(* CODESYS project e!C_SmartCoupler_Test_1.ecp

Project tree, tasks and I/O mapping:
  Generic_MODBUS_Master : ThirdParty Modbus Master, WAGO, order no. GenericModbusMaster, version 1.0.0.1
  PFCx00_SmartCoupler : 750-8202 PFC200 2ETH RS, WAGO, order no. 0750-8202, version 5.13.2.22
    application PFCx00_SmartCoupler
      libraries: ; VisuDialogs, * (System); WagoTypesCommon, 1.5.3.0 (WAGO); WagoAppHART, 1.7.1.0 (WAGO); WagoAppSolenoid, 1.7.1.0 (WAGO); WagoAppPowerMeasurement, 1.7.1.0 (WAGO); WagoTypesCom, 1.6.1.0 (WAGO); WagoAppDALI, 1.3.0.0 (WAGO); WagoSysKbusModule, 1.8.2.0 (WAGO); AnyViz Cloud Adapter, 1.4.0.0 (Mirasoft GmbH & Co. KG); WagoSysKbusServices, 1.8.7.0 (WAGO); WagoAppPlcModbus, 1.1.2.0 (WAGO); WagoTypesAsync_Internal_Template, 1.0.0.1 (WAGO); WagoSysModule_75x_632, 1.8.1.0 (WAGO); WagoSysModule_75x_48x, 1.5.1.0 (WAGO); WagoVisuIcons, 1.0.1.0 (WAGO); WagoSysModule_75x_49x, 1.7.1.0 (WAGO); WagoSysModule_753_647, 1.1.1.0 (WAGO); WagoAppKNX, 1.0.4.0 (WAGO)
      task Cloud_Task (freewheeling, priority 15) calls Cloud
      task PLC_Task (cyclic, interval t#10ms, priority 12) calls PLC_PRG
      task VISU_TASK (cyclic, interval 100 ms, priority 14) calls VisuElems.Visu_Prg
      program PLC_PRG [ST]
      GlobalData/
        global variables GCL_SmartCoupler
        global variables GVL_SmartCoupler
      Symbols
      visualisation Visualization
      program Cloud [ST]
    Kbus : Kbus, WAGO, version 1.4.0.2
        unmapped channels: K-BUS diagnostics
    MODBUS
      MODBUS : MODBUS, WAGO, order no. n/a, version 1.1.1.15
        LocalDeviceModbus : MODBUS Slave, WAGO, order no. n/a, version 1.1.1.15
          TcpSettings : Modbus TCP Slave, WAGO, order no. n/a, version 1.1.1.15
              settings: TCP Port = 503; TCP connection watchdog = 200 10ms
          UdpSettings : Modbus UDP Slave, WAGO, order no. n/a, version 1.1.1.15
              settings: UDP Port = 503
    Serial
      COM1 : COM1, WAGO, version 0.0.0.19
  libraries: WagoAppPlcModbus, * (WAGO); WagoAppHART, * (WAGO); WagoAppSolenoid, * (WAGO); WagoAppPowerMeasurement, * (WAGO); WagoTypesCom, * (WAGO); WagoTypesCommon, * (WAGO); WagoAppDALI, * (WAGO); VisuSymbols, 3.5.10.0 (System); WagoSysKbusModule, * (WAGO); WagoAppKNX, 1.0.4.0 (WAGO); WagoSysKbusServices, 1.8.7.0 (WAGO); WagoTypesAsync_Internal_Template, 1.0.0.1 (WAGO); WagoSysModule_75x_632, 1.8.1.0 (WAGO); WagoSysModule_75x_48x, 1.5.1.0 (WAGO); WagoVisuIcons, 1.0.1.0 (WAGO); WagoSysModule_75x_49x, 1.7.1.0 (WAGO); WagoSysModule_753_647, 1.1.1.0 (WAGO)
  GlobalStruct/
    data type DUT_WordAndBytes
    data type DUT_ModuleDataAccess
    data type DUT_RealAndBytes
    data type DUT_ModuleFunctionAccess
    data type DUT_ModuleDescriptor
    data type DUT_ModuleInterface
  GlobalProgram/
    program SmartCoupler [ST]: DrivePMeasurementModuleAccess, DriveSimpleDIOModuleAccess, DriveSolenoidModuleAccess, DriveHartModuleAccess, InitModuleDescriptor, DriveDaliModuleAccess, DriveSimpleAIOModuleAccess, DriveKnxModuleAccess
    program ModbusSlave [ST]: MapModbusData
  text list GlobalTextList
*)

// GlobalStruct/DUT_WordAndBytes
TYPE DUT_WordAndBytes :
UNION
	wValue: WORD;
	abValue: ARRAY[0..1] OF BYTE;	
END_UNION
END_TYPE

// GlobalStruct/DUT_ModuleDataAccess
TYPE DUT_ModuleDataAccess :
STRUCT
	sModuleList: STRING;
	udiModuleID: UDINT;
	auiOrderNumber: ARRAY[0..3] OF UINT;
	uiModuleChannels: UINT;
	uiModuleType: UINT;
	uiModulePiSize: UINT;
	uiModulePiInputSize: UINT;
	uiModulePiOutputSize: UINT;
	wModuleOutput_Data_1: WORD;
	wModuleOutput_Data_2: WORD;
	wModuleOutput_Data_3: WORD;
	wModuleOutput_Data_4: WORD;
	wModuleOutput_Data_5: WORD;
	wModuleOutput_Data_6: WORD;
	wModuleOutput_Data_7: WORD;
	wModuleOutput_Data_8: WORD;
	wModuleOutput_Data_9: WORD;
	wModuleOutput_Data_10: WORD;
	wModuleOutput_Data_11: WORD;
	wModuleOutput_Data_12: WORD;
	wModuleOutput_Data_13: WORD;
	wModuleOutput_Data_14: WORD;
	wModuleOutput_Data_15: WORD;
	wModuleOutput_Data_16: WORD;
	wModuleInput_Data_1: WORD;
	wModuleInput_Data_2: WORD;
	wModuleInput_Data_3: WORD;
	wModuleInput_Data_4: WORD;
	wModuleInput_Data_5: WORD;
	wModuleInput_Data_6: WORD;
	wModuleInput_Data_7: WORD;
	wModuleInput_Data_8: WORD;
	wModuleInput_Data_9: WORD;
	wModuleInput_Data_10: WORD;
	wModuleInput_Data_11: WORD;
	wModuleInput_Data_12: WORD;
	wModuleInput_Data_13: WORD;
	wModuleInput_Data_14: WORD;
	wModuleInput_Data_15: WORD;
	wModuleInput_Data_16: WORD;
	pawModuleOutput: POINTER TO ARRAY[1..GCL_SmartCoupler.LIM_OF_IO_FRAME] OF WORD;
	pawModuleInput: POINTER TO ARRAY[1..GCL_SmartCoupler.LIM_OF_IO_FRAME] OF WORD;
END_STRUCT
END_TYPE

// GlobalStruct/DUT_RealAndBytes
TYPE DUT_RealAndBytes :
UNION
	rValue: REAL;
	dwValue: DWORD;
	awValue: ARRAY[0..1] OF WORD;
	abValue: ARRAY[0..3] OF BYTE;
END_UNION
END_TYPE

// GlobalStruct/DUT_ModuleFunctionAccess
TYPE DUT_ModuleFunctionAccess :
STRUCT
	FbAC_Compact_494: WagoAppPowerMeasurement.FbAC_Compact_494;
	FbAC_Compact_495: WagoAppPowerMeasurement.FbAC_Compact_495;
	FbSolenoidBasicControl: WagoAppSolenoid.FbBasicControl;
	FbKnxMaster_TM: WagoAppKnx.FbKNX_Master_TM;
	FbDaliMaster: WagoAppDali.FbDaliMaster;
	FbDaliSendDimValue: WagoAppDali.FbDaliSendDimValue;
	FbHART_Current: WagoAppHart.FbHART_Current := (xEnable := TRUE);
	FbHART_CMD3_1: WagoAppHart.FbHART_CMD3;
	FbHART_CMD3_2: WagoAppHart.FbHART_CMD3;
	xHartReadTrigger_1: BOOL;
	xHartReadTrigger_2: BOOL;
	wHartChannelSchedule: WORD;
	TON_HartScheduleDelay: TON;
	TOF_HartCmdMonitor_1: TOF;
	TOF_HartCmdMonitor_2: TOF;
	tHartScheduleDelay: TIME := T#2S;
	tHartCmdMonitorTimeout: TIME := T#5S;
	iHartGenericErrorCnt: INT;
	iHartCmdErrorCnt_1: INT;
	iHartCmdErrorCnt_2: INT;
END_STRUCT
END_TYPE

// GlobalStruct/DUT_ModuleDescriptor
TYPE DUT_ModuleDescriptor :
STRUCT
	pDUT_ModuleInterface: POINTER TO DUT_ModuleInterface;
	pDUT_ModuleAccess: POINTER TO DUT_ModuleDataAccess;	
	pDUT_FunctionAccess: POINTER TO DUT_ModuleFunctionAccess;
END_STRUCT
END_TYPE

// GlobalStruct/DUT_ModuleInterface
TYPE DUT_ModuleInterface :
STRUCT
	FbModuleProcessInputsOutputs: WagoSysKbusModule.FbModuleProcessInputsOutputs;
	FbModule_75x_632: WagoSysKbusModule.FbModule_75x_632;
	FbModule_753_646: WagoSysKbusModule.FbModule_753_646;
	FbModule_753_647: WagoSysKbusModule.FbModule_753_647;
	FbModule_75x_48x: WagoSysKbusModule.FbModule_75x_48x;
	FbModule_75x_494: WagoSysKbusModule.FbModule_75x_494;
	FbModule_75x_495: WagoSysKbusModule.FbModule_75x_495;
(*
	FbModule_75x_632: WagoSysKbusModule.WagoSysModule_75x_632.FbModule_75x_632;
	FbModule_753_646: WagoSysKbusModule.WagoSysModule_753_646.FbModule_753_646;
	FbModule_753_647: WagoSysKbusModule.WagoSysModule_753_647.FbModule_753_647;
	FbModule_75x_48x: WagoSysKbusModule.WagoSysModule_75x_48x.FbModule_75x_48x;
	FbModule_75x_494: WagoSysKbusModule.WagoSysModule_75x_49x.FbModule_75x_494;
	FbModule_75x_495: WagoSysKbusModule.WagoSysModule_75x_49x.FbModule_75x_495;
*)
END_STRUCT
END_TYPE

// PFCx00_SmartCoupler/PFCx00_SmartCoupler/GlobalData/GCL_SmartCoupler
{attribute 'qualified_only'}
VAR_GLOBAL CONSTANT
	LIM_OF_IO_MODULES: INT := 64;
	LIM_OF_IO_SEGMENT: INT := 4096;
	LIM_OF_IO_FRAME: USINT := 16; (* Number of WORD per module *)
END_VAR

// PFCx00_SmartCoupler/PFCx00_SmartCoupler/GlobalData/GVL_SmartCoupler
{attribute 'qualified_only'}
VAR_GLOBAL
	aDUT_ModuleDescriptor: ARRAY[1..GCL_SmartCoupler.LIM_OF_IO_MODULES] OF DUT_ModuleDescriptor;
	aDUT_ModuleInterface: ARRAY[1..GCL_SmartCoupler.LIM_OF_IO_MODULES] OF DUT_ModuleInterface;
	aDUT_ModuleDataAccess: ARRAY[1..GCL_SmartCoupler.LIM_OF_IO_MODULES] OF DUT_ModuleDataAccess;
	aDUT_ModuleFunctionAccess: ARRAY[1..GCL_SmartCoupler.LIM_OF_IO_MODULES] OF DUT_ModuleFunctionAccess;	
	awModuleInputData: ARRAY[1..GCL_SmartCoupler.LIM_OF_IO_SEGMENT] OF WORD;
	awModuleOutputData: ARRAY[1..GCL_SmartCoupler.LIM_OF_IO_SEGMENT] OF WORD;
	DUT_ModuleData: DUT_RealAndBytes;
	bModule646Index: BYTE;
	bModule647Index: BYTE;
END_VAR

// PFCx00_SmartCoupler/PFCx00_SmartCoupler/Cloud
PROGRAM Cloud
VAR
	AnyVizClient: AnyVizClient := (ProjectID := 324, Password := 'wago1234');
	Status: STRING(255);
	Error: BOOL;
	Connected: BOOL;
END_VAR


(*
AnyVizClient(
	Status				=> Status, 
	Error				=> Error, 
	Connected			=> Connected);
*)

END_PROGRAM

// PFCx00_SmartCoupler/PFCx00_SmartCoupler/PLC_PRG
PROGRAM PLC_PRG
VAR

END_VAR



ModbusSlave();
SmartCoupler();

END_PROGRAM

// GlobalProgram/ModbusSlave
PROGRAM ModbusSlave
VAR
	FbMbSimpleServerUdp: FbMbSimpleServerUdp;
	FbMbSimpleServerTcp: FbMbSimpleServerTcp;
	xMbTcpOpen: BOOL := TRUE;
	wMbTcpPort: WORD := 502;
	utMbTcpKeepAlive: typKeepAlive;
	xMbTcpIsOpen: BOOL;
	xMbTcpError: BOOL;
	oMbTcpStatus: WagoSysErrorBase.FbResult;
	udiMbTcpConnectedClients: UDINT;
	bMbTcpUnitId: BYTE := 1;
	axMbDiscreteInputs: ARRAY[0..0] OF BOOL;
	axMbCoils: ARRAY[0..0] OF BOOL;
	oMbTcpAccessInfo: FbMbAccessInfo;
	xMbUdpOpen: BOOL := TRUE;
	wMbUdpPort: WORD := 502;
	xMbUdpIsOpen: BOOL;
	xMbUdpError: BOOL;
	oMbUdpStatus: WagoSysErrorBase.FbResult;
	bMbUdpUnitId: BYTE := 1;
	oMbUdpAccessInfo: FbMbAccessInfo;
	FbMbSimpleServerSerial: FbMbSimpleServerSerial;
	xMbRtuConnect: BOOL := TRUE;
	udiMbRtuBaudrate: UDINT := 19200;
	usiMbRtuDataBits: USINT := 8;
	eMbRtuParity: WagoTypesCom.eTTYParity := ETTYPARITY.None;
	eMbRtuStopBits: WagoTypesCom.eTTYStopBits := ETTYSTOPBITS.one;
	eMbRtuHandshake: WagoTypesCom.eTTYHandshake := ETTYHANDSHAKE.None;
	eMbRtuPhysical: WagoTypesCom.eTTYPhysicalLayer := ETTYPHYSICALLAYER.RS485_HalfDuplex;
	eMbRtuFrameType: eMbFrameType := EMBFRAMETYPE.RTU;
	xMbRtuIsConnected: BOOL;
	xMbRtuError: BOOL;
	oMbRtuStatus: WagoSysErrorBase.FbResult;
	bMbRtuUnitId: BYTE := 1;
	oMbRtuAccessInfo: FbMbAccessInfo;
END_VAR


FbMbSimpleServerTcp(
	xOpen				:= xMbTcpOpen, 
	wPort				:= wMbTcpPort, 
	utKeepAlive			:= utMbTcpKeepAlive, 
	xIsOpen				=> xMbTcpIsOpen, 
	xError				=> xMbTcpError, 
	oStatus				=> oMbTcpStatus, 
	udiConnectedClients	=> udiMbTcpConnectedClients, 
	bUnitId				:= bMbTcpUnitId, 
	axDiscreteInputs	:= axMbDiscreteInputs, 
	axCoils				:= axMbCoils, 
	awInputRegisters	:= GVL_SmartCoupler.awModuleInputData, 
	awHoldingRegisters	:= GVL_SmartCoupler.awModuleOutputData, 
	oMbAccessInfo		=> oMbTcpAccessInfo);

FbMbSimpleServerUdp(
	xOpen				:= xMbUdpOpen, 
	wPort				:= wMbUdpPort, 
	xIsOpen				=> xMbUdpIsOpen, 
	xError				=> xMbUdpError, 
	oStatus				=> oMbUdpStatus, 
	bUnitId				:= bMbUdpUnitId, 
	axDiscreteInputs	:= axMbDiscreteInputs, 
	axCoils				:= axMbCoils, 
	awInputRegisters	:= GVL_SmartCoupler.awModuleInputData, 
	awHoldingRegisters	:= GVL_SmartCoupler.awModuleOutputData, 
	oMbAccessInfo		=> oMbUdpAccessInfo);

FbMbSimpleServerSerial(
	xConnect			:= xMbRtuConnect, 
	I_Port				:= COM1, 
	udiBaudrate			:= udiMbRtuBaudrate, 
	usiDataBits			:= usiMbRtuDataBits, 
	eParity				:= eMbRtuParity, 
	eStopBits			:= eMbRtuStopBits, 
	eHandshake			:= eMbRtuHandshake, 
	ePhysical			:= eMbRtuPhysical, 
	eFrameType			:= eMbRtuFrameType, 
	xIsConnected		=> xMbRtuIsConnected, 
	xError				=> xMbRtuError, 
	oStatus				=> oMbRtuStatus, 
	bUnitId				:= bMbRtuUnitId, 
	axDiscreteInputs	:= axMbDiscreteInputs, 
	axCoils				:= axMbCoils, 
	awInputRegisters	:= GVL_SmartCoupler.awModuleInputData, 
	awHoldingRegisters	:= GVL_SmartCoupler.awModuleOutputData, 
	oMbAccessInfo		=> oMbRtuAccessInfo);

ACTION MapModbusData:

;
END_ACTION

END_PROGRAM

// GlobalProgram/SmartCoupler
PROGRAM SmartCoupler
VAR
	I_Terminal: WagoSysModuleBase.WagoTypesModuleBase.I_TerminalBase;
	FBTerminalManagerResult: FBResult;
	xTerminalInit: BOOL;
	usiModuleIndex: USINT;
	uiModuleMapIndex: UINT;
	usiModuleIndexLimit: USINT;
	uiChannelIndex: UINT;
END_VAR


IF  (TerminalManager.isBusInit(WagoTypesBusServices.eBusType.KBUS) = TRUE) THEN
	IF (xTerminalInit = FALSE) THEN
		usiModuleIndexLimit := TerminalManager.getTerminalQuantity(WagoSysKbusModule.KBUS);
	END_IF
	uiModuleMapIndex := 1;
	GVL_SmartCoupler.bModule646Index := 1;
	GVL_SmartCoupler.bModule647Index := 1;
	FOR usiModuleIndex := 1 TO usiModuleIndexLimit DO
		GVL_SmartCoupler.aDUT_ModuleDescriptor[usiModuleIndex].pDUT_ModuleInterface := ADR(GVL_SmartCoupler.aDUT_ModuleInterface[usiModuleIndex]);
		GVL_SmartCoupler.aDUT_ModuleDescriptor[usiModuleIndex].pDUT_ModuleAccess := ADR(GVL_SmartCoupler.aDUT_ModuleDataAccess[usiModuleIndex]);
		GVL_SmartCoupler.aDUT_ModuleDescriptor[usiModuleIndex].pDUT_FunctionAccess := ADR(GVL_SmartCoupler.aDUT_ModuleFunctionAccess[usiModuleIndex]);
		IF (xTerminalInit = FALSE) THEN
			InitModuleDescriptor();
		ELSE
	
			(* Data exchange for Address-based fieldbus interface/gateway, e.g. Modbus *)
			GVL_SmartCoupler.aDUT_ModuleDataAccess[usiModuleIndex].pawModuleInput := ADR(GVL_SmartCoupler.awModuleInputData[uiModuleMapIndex]);
			GVL_SmartCoupler.aDUT_ModuleDataAccess[usiModuleIndex].pawModuleOutput := ADR(GVL_SmartCoupler.awModuleOutputData[uiModuleMapIndex]);

			(* Data exchange for Symbol-based fieldbus interface/gateway, e.g. OPCUA *)
			(*
			GVL_SmartCoupler.aDUT_ModuleDataAccess[usiModuleIndex].pawModuleInput := ADR(GVL_SmartCoupler.aDUT_ModuleDataAccess[usiModuleIndex].wModuleInput_Data_1);
			GVL_SmartCoupler.aDUT_ModuleDataAccess[usiModuleIndex].pawModuleOutput := ADR(GVL_SmartCoupler.aDUT_ModuleDataAccess[usiModuleIndex].wModuleOutput_Data_1);
			*)
			CASE GVL_SmartCoupler.aDUT_ModuleDataAccess[usiModuleIndex].uiModuleType OF
	
				COMPLEX_INPUT, COMPLEX_OUTPUT:
					DriveSimpleAIOModuleAccess();
				COMPLEX_INOUT:
					CASE GVL_SmartCoupler.aDUT_ModuleDataAccess[usiModuleIndex].auiOrderNumber[1] OF
						482, 484:
							DriveHartModuleAccess();
						494, 495:
							DrivePMeasurementModuleAccess();
						632:
							DriveSolenoidModuleAccess();
						646:
							DriveKnxModuleAccess();
							GVL_SmartCoupler.bModule646Index := GVL_SmartCoupler.bModule646Index + 1;
						647:
							DriveDaliModuleAccess();
							GVL_SmartCoupler.bModule647Index := GVL_SmartCoupler.bModule647Index + 1;
					END_CASE
				DIGITAL_INPUT, DIGITAL_INPUT_DIAG, DIGITAL_OUTPUT, DIGITAL_OUTPUT_DIAG, DIGITAL_INOUT, DIGITAL_INOUT_DIAG, DIGITAL_DIAG:
					DriveSimpleDIOModuleAccess();
	
			END_CASE
			uiModuleMapIndex := uiModuleMapIndex + GCL_SmartCoupler.LIM_OF_IO_FRAME;
		END_IF
	END_FOR
	xTerminalInit := TRUE;
END_IF

ACTION DrivePMeasurementModuleAccess:

IF (GVL_SmartCoupler.aDUT_ModuleDataAccess[usiModuleIndex].uiModuleType = 494) THEN
	GVL_SmartCoupler.aDUT_ModuleFunctionAccess[usiModuleIndex].FbAC_Compact_494.xEnable (*:= WORD_TO_BOOL(GVL_SmartCoupler.aDUT_ModuleDataAccess[usiModuleIndex].pawModuleOutput^[1])*);
	GVL_SmartCoupler.aDUT_ModuleFunctionAccess[usiModuleIndex].FbAC_Compact_494.tCycleTime (*:= WORD_TO_TIME(GVL_SmartCoupler.aDUT_ModuleDataAccess[usiModuleIndex].pawModuleOutput^[2])*);
	GVL_SmartCoupler.aDUT_ModuleFunctionAccess[usiModuleIndex].FbAC_Compact_494.rSelectedScalingFactor (*:= WORD_TO_REAL(GVL_SmartCoupler.aDUT_ModuleDataAccess[usiModuleIndex].pawModuleOutput^[3])*);	
	GVL_SmartCoupler.aDUT_ModuleFunctionAccess[usiModuleIndex].FbAC_Compact_494(I_Port := GVL_SmartCoupler.aDUT_ModuleInterface[usiModuleIndex].FbModule_75x_494);
	GVL_SmartCoupler.DUT_ModuleData.rValue := GVL_SmartCoupler.aDUT_ModuleFunctionAccess[usiModuleIndex].FbAC_Compact_494.aVoltage_L_N[1];
	GVL_SmartCoupler.aDUT_ModuleDataAccess[usiModuleIndex].pawModuleInput^[1] := GVL_SmartCoupler.DUT_ModuleData.awValue[0];
	GVL_SmartCoupler.aDUT_ModuleDataAccess[usiModuleIndex].pawModuleInput^[2] := GVL_SmartCoupler.DUT_ModuleData.awValue[1];
	GVL_SmartCoupler.DUT_ModuleData.rValue := GVL_SmartCoupler.aDUT_ModuleFunctionAccess[usiModuleIndex].FbAC_Compact_494.aVoltage_L_N[2];
	GVL_SmartCoupler.aDUT_ModuleDataAccess[usiModuleIndex].pawModuleInput^[3] := GVL_SmartCoupler.DUT_ModuleData.awValue[0];
	GVL_SmartCoupler.aDUT_ModuleDataAccess[usiModuleIndex].pawModuleInput^[4] := GVL_SmartCoupler.DUT_ModuleData.awValue[1];
	GVL_SmartCoupler.DUT_ModuleData.rValue := GVL_SmartCoupler.aDUT_ModuleFunctionAccess[usiModuleIndex].FbAC_Compact_494.aVoltage_L_N[3];
	GVL_SmartCoupler.aDUT_ModuleDataAccess[usiModuleIndex].pawModuleInput^[5] := GVL_SmartCoupler.DUT_ModuleData.awValue[0];
	GVL_SmartCoupler.aDUT_ModuleDataAccess[usiModuleIndex].pawModuleInput^[6] := GVL_SmartCoupler.DUT_ModuleData.awValue[1];
ELSIF (GVL_SmartCoupler.aDUT_ModuleDataAccess[usiModuleIndex].uiModuleType = 495) THEN
	GVL_SmartCoupler.aDUT_ModuleFunctionAccess[usiModuleIndex].FbAC_Compact_495.xEnable (*:= WORD_TO_BOOL(GVL_SmartCoupler.aDUT_ModuleDataAccess[usiModuleIndex].pawModuleOutput^[1])*);
	GVL_SmartCoupler.aDUT_ModuleFunctionAccess[usiModuleIndex].FbAC_Compact_495.tCycleTime (*:= WORD_TO_TIME(GVL_SmartCoupler.aDUT_ModuleDataAccess[usiModuleIndex].pawModuleOutput^[2])*);
	GVL_SmartCoupler.aDUT_ModuleFunctionAccess[usiModuleIndex].FbAC_Compact_495.rSelectedScalingFactor (*:= WORD_TO_REAL(GVL_SmartCoupler.aDUT_ModuleDataAccess[usiModuleIndex].pawModuleOutput^[3])*);
	GVL_SmartCoupler.aDUT_ModuleFunctionAccess[usiModuleIndex].FbAC_Compact_495(I_Port := GVL_SmartCoupler.aDUT_ModuleInterface[usiModuleIndex].FbModule_75x_495);
	GVL_SmartCoupler.DUT_ModuleData.rValue := GVL_SmartCoupler.aDUT_ModuleFunctionAccess[usiModuleIndex].FbAC_Compact_495.aVoltage_L_N[1];
	GVL_SmartCoupler.aDUT_ModuleDataAccess[usiModuleIndex].pawModuleInput^[1] := GVL_SmartCoupler.DUT_ModuleData.awValue[0];
	GVL_SmartCoupler.aDUT_ModuleDataAccess[usiModuleIndex].pawModuleInput^[2] := GVL_SmartCoupler.DUT_ModuleData.awValue[1];
	GVL_SmartCoupler.DUT_ModuleData.rValue := GVL_SmartCoupler.aDUT_ModuleFunctionAccess[usiModuleIndex].FbAC_Compact_495.aVoltage_L_N[2];
	GVL_SmartCoupler.aDUT_ModuleDataAccess[usiModuleIndex].pawModuleInput^[3] := GVL_SmartCoupler.DUT_ModuleData.awValue[0];
	GVL_SmartCoupler.aDUT_ModuleDataAccess[usiModuleIndex].pawModuleInput^[4] := GVL_SmartCoupler.DUT_ModuleData.awValue[1];
	GVL_SmartCoupler.DUT_ModuleData.rValue := GVL_SmartCoupler.aDUT_ModuleFunctionAccess[usiModuleIndex].FbAC_Compact_495.aVoltage_L_N[3];
	GVL_SmartCoupler.aDUT_ModuleDataAccess[usiModuleIndex].pawModuleInput^[5] := GVL_SmartCoupler.DUT_ModuleData.awValue[0];
	GVL_SmartCoupler.aDUT_ModuleDataAccess[usiModuleIndex].pawModuleInput^[6] := GVL_SmartCoupler.DUT_ModuleData.awValue[1];
END_IF
END_ACTION

ACTION DriveSimpleDIOModuleAccess:

FOR uiChannelIndex := 0 TO GVL_SmartCoupler.aDUT_ModuleDataAccess[usiModuleIndex].uiModuleChannels DO
	IF (GVL_SmartCoupler.aDUT_ModuleDataAccess[usiModuleIndex].uiModulePiInputSize > 0) THEN
		GVL_SmartCoupler.aDUT_ModuleDataAccess[usiModuleIndex].pawModuleInput^[uiChannelIndex+1] :=
			BOOL_TO_WORD(
				GVL_SmartCoupler.aDUT_ModuleInterface[usiModuleIndex].FbModuleProcessInputsOutputs.GetProcessInBit(
							ByteNo	:= 0,
							BitNo	:= UINT_TO_USINT(uiChannelIndex)));
	END_IF
	IF (GVL_SmartCoupler.aDUT_ModuleDataAccess[usiModuleIndex].uiModulePiOutputSize > 0) THEN
		GVL_SmartCoupler.aDUT_ModuleInterface[usiModuleIndex].FbModuleProcessInputsOutputs.SetProcessOutBit(
			ByteNo	:= 0,
			BitNo	:= UINT_TO_USINT(uiChannelIndex),
			OutData	:= WORD_TO_BOOL(GVL_SmartCoupler.aDUT_ModuleDataAccess[usiModuleIndex].pawModuleOutput^[uiChannelIndex+1]));
	END_IF
END_FOR
END_ACTION

ACTION DriveSolenoidModuleAccess:

GVL_SmartCoupler.aDUT_ModuleFunctionAccess[usiModuleIndex].FbSolenoidBasicControl.bSolenoidNo := WORD_TO_BYTE(GVL_SmartCoupler.aDUT_ModuleDataAccess[usiModuleIndex].pawModuleOutput^[1]);
GVL_SmartCoupler.aDUT_ModuleFunctionAccess[usiModuleIndex].FbSolenoidBasicControl.xPowerEnable := WORD_TO_BOOL(GVL_SmartCoupler.aDUT_ModuleDataAccess[usiModuleIndex].pawModuleOutput^[2]);
GVL_SmartCoupler.aDUT_ModuleFunctionAccess[usiModuleIndex].FbSolenoidBasicControl.xCurrentEnable := WORD_TO_BOOL(GVL_SmartCoupler.aDUT_ModuleDataAccess[usiModuleIndex].pawModuleOutput^[3]);
GVL_SmartCoupler.aDUT_ModuleFunctionAccess[usiModuleIndex].FbSolenoidBasicControl.xDitherEnable := WORD_TO_BOOL(GVL_SmartCoupler.aDUT_ModuleDataAccess[usiModuleIndex].pawModuleOutput^[4]);
GVL_SmartCoupler.aDUT_ModuleFunctionAccess[usiModuleIndex].FbSolenoidBasicControl.iCurrent := WORD_TO_INT(GVL_SmartCoupler.aDUT_ModuleDataAccess[usiModuleIndex].pawModuleOutput^[5]);

GVL_SmartCoupler.aDUT_ModuleFunctionAccess[usiModuleIndex].FbSolenoidBasicControl(I_Port := GVL_SmartCoupler.aDUT_ModuleInterface[usiModuleIndex].FbModule_75x_632);

IF (GVL_SmartCoupler.aDUT_ModuleFunctionAccess[usiModuleIndex].FbSolenoidBasicControl.bSolenoidNo = 1) THEN
	GVL_SmartCoupler.aDUT_ModuleDataAccess[usiModuleIndex].pawModuleInput^[1] := INT_TO_WORD(GVL_SmartCoupler.aDUT_ModuleFunctionAccess[usiModuleIndex].FbSolenoidBasicControl.iActualCurrent);
	GVL_SmartCoupler.aDUT_ModuleDataAccess[usiModuleIndex].pawModuleInput^[2] := BOOL_TO_WORD(GVL_SmartCoupler.aDUT_ModuleFunctionAccess[usiModuleIndex].FbSolenoidBasicControl.xEnabled);
	GVL_SmartCoupler.aDUT_ModuleDataAccess[usiModuleIndex].pawModuleInput^[3] := BOOL_TO_WORD(GVL_SmartCoupler.aDUT_ModuleFunctionAccess[usiModuleIndex].FbSolenoidBasicControl.xError);
ELSIF (GVL_SmartCoupler.aDUT_ModuleFunctionAccess[usiModuleIndex].FbSolenoidBasicControl.bSolenoidNo = 2) THEN
	GVL_SmartCoupler.aDUT_ModuleDataAccess[usiModuleIndex].pawModuleInput^[9] := INT_TO_WORD(GVL_SmartCoupler.aDUT_ModuleFunctionAccess[usiModuleIndex].FbSolenoidBasicControl.iActualCurrent);
	GVL_SmartCoupler.aDUT_ModuleDataAccess[usiModuleIndex].pawModuleInput^[10] := BOOL_TO_WORD(GVL_SmartCoupler.aDUT_ModuleFunctionAccess[usiModuleIndex].FbSolenoidBasicControl.xEnabled);
	GVL_SmartCoupler.aDUT_ModuleDataAccess[usiModuleIndex].pawModuleInput^[11] := BOOL_TO_WORD(GVL_SmartCoupler.aDUT_ModuleFunctionAccess[usiModuleIndex].FbSolenoidBasicControl.xError);
END_IF
END_ACTION

ACTION DriveHartModuleAccess:

(*GVL_SmartCoupler.aDUT_ModuleFunctionAccess[usiModuleIndex].FbHART_Current.xEnable := WORD_TO_BOOL(GVL_SmartCoupler.aDUT_ModuleDataAccess[usiModuleIndex].pawModuleOutput^[1]);*)

GVL_SmartCoupler.aDUT_ModuleFunctionAccess[usiModuleIndex].FbHART_Current( 
	I_Port				:= GVL_SmartCoupler.aDUT_ModuleInterface[usiModuleIndex].FbModule_75x_48x);

GVL_SmartCoupler.DUT_ModuleData.rValue := GVL_SmartCoupler.aDUT_ModuleFunctionAccess[usiModuleIndex].FbHART_Current.rCurrentChannel_1;
GVL_SmartCoupler.aDUT_ModuleDataAccess[usiModuleIndex].pawModuleInput^[1] := GVL_SmartCoupler.DUT_ModuleData.awValue[0];
GVL_SmartCoupler.aDUT_ModuleDataAccess[usiModuleIndex].pawModuleInput^[2] := GVL_SmartCoupler.DUT_ModuleData.awValue[1];
GVL_SmartCoupler.aDUT_ModuleDataAccess[usiModuleIndex].pawModuleInput^[6] := GVL_SmartCoupler.aDUT_ModuleFunctionAccess[usiModuleIndex].FbHART_Current.wCurrent_1 AND 2#00000000_00000011;
GVL_SmartCoupler.aDUT_ModuleDataAccess[usiModuleIndex].pawModuleInput^[7] := INT_TO_WORD(GVL_SmartCoupler.aDUT_ModuleFunctionAccess[usiModuleIndex].iHartCmdErrorCnt_1);

GVL_SmartCoupler.DUT_ModuleData.rValue := GVL_SmartCoupler.aDUT_ModuleFunctionAccess[usiModuleIndex].FbHART_Current.rCurrentChannel_2;
GVL_SmartCoupler.aDUT_ModuleDataAccess[usiModuleIndex].pawModuleInput^[9] := GVL_SmartCoupler.DUT_ModuleData.awValue[0];
GVL_SmartCoupler.aDUT_ModuleDataAccess[usiModuleIndex].pawModuleInput^[10] := GVL_SmartCoupler.DUT_ModuleData.awValue[1];
GVL_SmartCoupler.aDUT_ModuleDataAccess[usiModuleIndex].pawModuleInput^[14] := GVL_SmartCoupler.aDUT_ModuleFunctionAccess[usiModuleIndex].FbHART_Current.wCurrent_2 AND 2#00000000_00000011;
GVL_SmartCoupler.aDUT_ModuleDataAccess[usiModuleIndex].pawModuleInput^[15] := INT_TO_WORD(GVL_SmartCoupler.aDUT_ModuleFunctionAccess[usiModuleIndex].iHartCmdErrorCnt_2);

CASE GVL_SmartCoupler.aDUT_ModuleFunctionAccess[usiModuleIndex].wHartChannelSchedule OF
	0:
		GVL_SmartCoupler.aDUT_ModuleFunctionAccess[usiModuleIndex].TON_HartScheduleDelay(IN:= TRUE, PT:= GVL_SmartCoupler.aDUT_ModuleFunctionAccess[usiModuleIndex].tHartScheduleDelay);
		IF (GVL_SmartCoupler.aDUT_ModuleFunctionAccess[usiModuleIndex].TON_HartScheduleDelay.Q = TRUE) THEN
			GVL_SmartCoupler.aDUT_ModuleFunctionAccess[usiModuleIndex].TON_HartScheduleDelay(IN:= FALSE);
			GVL_SmartCoupler.aDUT_ModuleFunctionAccess[usiModuleIndex].wHartChannelSchedule := 1;
		END_IF
	1:
		IF (GVL_SmartCoupler.aDUT_ModuleFunctionAccess[usiModuleIndex].FbHART_Current.xError = TRUE) THEN
			GVL_SmartCoupler.aDUT_ModuleFunctionAccess[usiModuleIndex].wHartChannelSchedule := 1000;
		ELSE
			GVL_SmartCoupler.aDUT_ModuleFunctionAccess[usiModuleIndex].xHartReadTrigger_1 := TRUE;
			GVL_SmartCoupler.aDUT_ModuleFunctionAccess[usiModuleIndex].wHartChannelSchedule := 10;
		END_IF

	10:
		GVL_SmartCoupler.aDUT_ModuleFunctionAccess[usiModuleIndex].FbHART_CMD3_1(
			I_Port	:= GVL_SmartCoupler.aDUT_ModuleInterface[usiModuleIndex].FbModule_75x_48x, 
			bChannel:= 1, 
			xTrigger:= GVL_SmartCoupler.aDUT_ModuleFunctionAccess[usiModuleIndex].xHartReadTrigger_1);
			GVL_SmartCoupler.DUT_ModuleData.rValue := GVL_SmartCoupler.aDUT_ModuleFunctionAccess[usiModuleIndex].FbHART_CMD3_1.typData.rVarPrimary;
			GVL_SmartCoupler.aDUT_ModuleDataAccess[usiModuleIndex].pawModuleInput^[3] := GVL_SmartCoupler.DUT_ModuleData.awValue[0];
			GVL_SmartCoupler.aDUT_ModuleDataAccess[usiModuleIndex].pawModuleInput^[4] := GVL_SmartCoupler.DUT_ModuleData.awValue[1];
			IF ((GVL_SmartCoupler.aDUT_ModuleFunctionAccess[usiModuleIndex].FbHART_Current.wCurrent_1 AND 2#00000000_00000011) <>  2#00000000_00000000) THEN
				GVL_SmartCoupler.aDUT_ModuleFunctionAccess[usiModuleIndex].TOF_HartCmdMonitor_1(IN:= FALSE);
				GVL_SmartCoupler.aDUT_ModuleDataAccess[usiModuleIndex].pawModuleInput^[5] := 0;
			ELSE
				GVL_SmartCoupler.aDUT_ModuleFunctionAccess[usiModuleIndex].TOF_HartCmdMonitor_1(IN:= GVL_SmartCoupler.aDUT_ModuleFunctionAccess[usiModuleIndex].FbHART_CMD3_1.xError, PT:= GVL_SmartCoupler.aDUT_ModuleFunctionAccess[usiModuleIndex].tHartCmdMonitorTimeout);
				GVL_SmartCoupler.aDUT_ModuleDataAccess[usiModuleIndex].pawModuleInput^[5] := BOOL_TO_WORD(GVL_SmartCoupler.aDUT_ModuleFunctionAccess[usiModuleIndex].TOF_HartCmdMonitor_1.Q);
				IF (GVL_SmartCoupler.aDUT_ModuleFunctionAccess[usiModuleIndex].FbHART_CMD3_1.xError = TRUE) THEN
					GVL_SmartCoupler.aDUT_ModuleFunctionAccess[usiModuleIndex].iHartCmdErrorCnt_1 := GVL_SmartCoupler.aDUT_ModuleFunctionAccess[usiModuleIndex].iHartCmdErrorCnt_1 + 1;
				END_IF
			END_IF
		IF (GVL_SmartCoupler.aDUT_ModuleFunctionAccess[usiModuleIndex].xHartReadTrigger_1 = FALSE) THEN
			GVL_SmartCoupler.aDUT_ModuleFunctionAccess[usiModuleIndex].xHartReadTrigger_2 := TRUE;
			GVL_SmartCoupler.aDUT_ModuleFunctionAccess[usiModuleIndex].wHartChannelSchedule := 20;
		END_IF
	20:
		GVL_SmartCoupler.aDUT_ModuleFunctionAccess[usiModuleIndex].FbHART_CMD3_2(
			I_Port	:= GVL_SmartCoupler.aDUT_ModuleInterface[usiModuleIndex].FbModule_75x_48x, 
			bChannel:= 2, 
			xTrigger:= GVL_SmartCoupler.aDUT_ModuleFunctionAccess[usiModuleIndex].xHartReadTrigger_2);
			GVL_SmartCoupler.DUT_ModuleData.rValue := GVL_SmartCoupler.aDUT_ModuleFunctionAccess[usiModuleIndex].FbHART_CMD3_2.typData.rVarPrimary;
			GVL_SmartCoupler.aDUT_ModuleDataAccess[usiModuleIndex].pawModuleInput^[11] := GVL_SmartCoupler.DUT_ModuleData.awValue[0];
			GVL_SmartCoupler.aDUT_ModuleDataAccess[usiModuleIndex].pawModuleInput^[12] := GVL_SmartCoupler.DUT_ModuleData.awValue[1];
			IF ((GVL_SmartCoupler.aDUT_ModuleFunctionAccess[usiModuleIndex].FbHART_Current.wCurrent_2 AND 2#00000000_00000011) <>  2#00000000_00000000) THEN
				GVL_SmartCoupler.aDUT_ModuleFunctionAccess[usiModuleIndex].TOF_HartCmdMonitor_2(IN:= FALSE);
				GVL_SmartCoupler.aDUT_ModuleDataAccess[usiModuleIndex].pawModuleInput^[13] := 0;
			ELSE
				GVL_SmartCoupler.aDUT_ModuleFunctionAccess[usiModuleIndex].TOF_HartCmdMonitor_2(IN:= GVL_SmartCoupler.aDUT_ModuleFunctionAccess[usiModuleIndex].FbHART_CMD3_2.xError, PT:= GVL_SmartCoupler.aDUT_ModuleFunctionAccess[usiModuleIndex].tHartCmdMonitorTimeout);
				GVL_SmartCoupler.aDUT_ModuleDataAccess[usiModuleIndex].pawModuleInput^[13] := BOOL_TO_WORD(GVL_SmartCoupler.aDUT_ModuleFunctionAccess[usiModuleIndex].TOF_HartCmdMonitor_2.Q);
				IF (GVL_SmartCoupler.aDUT_ModuleFunctionAccess[usiModuleIndex].FbHART_CMD3_2.xError = TRUE) THEN
					GVL_SmartCoupler.aDUT_ModuleFunctionAccess[usiModuleIndex].iHartCmdErrorCnt_2 := GVL_SmartCoupler.aDUT_ModuleFunctionAccess[usiModuleIndex].iHartCmdErrorCnt_2 + 1;
				END_IF				
			END_IF
		IF (GVL_SmartCoupler.aDUT_ModuleFunctionAccess[usiModuleIndex].xHartReadTrigger_2 = FALSE) THEN
			GVL_SmartCoupler.aDUT_ModuleFunctionAccess[usiModuleIndex].wHartChannelSchedule := 0;
		END_IF

	1000: (* Error Handling...*)
		GVL_SmartCoupler.aDUT_ModuleFunctionAccess[usiModuleIndex].FbHART_Current.xEnable := FALSE;
		GVL_SmartCoupler.aDUT_ModuleFunctionAccess[usiModuleIndex].iHartGenericErrorCnt := GVL_SmartCoupler.aDUT_ModuleFunctionAccess[usiModuleIndex].iHartGenericErrorCnt + 1;
		GVL_SmartCoupler.aDUT_ModuleFunctionAccess[usiModuleIndex].wHartChannelSchedule := 1001;
	1001:
		GVL_SmartCoupler.aDUT_ModuleFunctionAccess[usiModuleIndex].FbHART_Current.xEnable := TRUE;
		GVL_SmartCoupler.aDUT_ModuleFunctionAccess[usiModuleIndex].wHartChannelSchedule := 0;		

END_CASE
END_ACTION

ACTION InitModuleDescriptor:

I_Terminal := TerminalManager.getTerminalBySlotNo(WagoTypesBusServices.eBusType.KBUS,usiModuleIndex);
GVL_SmartCoupler.aDUT_ModuleDataAccess[usiModuleIndex].sModuleList 		:= I_Terminal.getOrderNumberAsString();
GVL_SmartCoupler.aDUT_ModuleDataAccess[usiModuleIndex].uiModuleChannels	:= I_Terminal.getChannels();
GVL_SmartCoupler.aDUT_ModuleDataAccess[usiModuleIndex].uiModuleType		:= I_Terminal.getModuleType();
GVL_SmartCoupler.aDUT_ModuleDataAccess[usiModuleIndex].uiModulePiSize	:= I_Terminal.getPaSize();
GVL_SmartCoupler.aDUT_ModuleDataAccess[usiModuleIndex].udiModuleID		:= I_Terminal.getModuleId();
GVL_SmartCoupler.aDUT_ModuleDataAccess[usiModuleIndex].auiOrderNumber	:= I_Terminal.getOrderNumber();

CASE GVL_SmartCoupler.aDUT_ModuleDataAccess[usiModuleIndex].uiModuleType OF

	COMPLEX_INOUT:
		CASE GVL_SmartCoupler.aDUT_ModuleDataAccess[usiModuleIndex].auiOrderNumber[1] OF
			482,484:
				TerminalManager.RegisterModuleAtTerminal(GVL_SmartCoupler.aDUT_ModuleInterface[usiModuleIndex].FbModule_75x_48x,I_Terminal);
			494:
				TerminalManager.RegisterModuleAtTerminal(GVL_SmartCoupler.aDUT_ModuleInterface[usiModuleIndex].FbModule_75x_494,I_Terminal);
			495:
				TerminalManager.RegisterModuleAtTerminal(GVL_SmartCoupler.aDUT_ModuleInterface[usiModuleIndex].FbModule_75x_495,I_Terminal);
			632:
				TerminalManager.RegisterModuleAtTerminal(GVL_SmartCoupler.aDUT_ModuleInterface[usiModuleIndex].FbModule_75x_632,I_Terminal);
			646:
				TerminalManager.RegisterModuleAtTerminal(GVL_SmartCoupler.aDUT_ModuleInterface[usiModuleIndex].FbModule_753_646,I_Terminal);
			647:
				TerminalManager.RegisterModuleAtTerminal(GVL_SmartCoupler.aDUT_ModuleInterface[usiModuleIndex].FbModule_753_647,I_Terminal);
		END_CASE

	COMPLEX_INPUT, COMPLEX_OUTPUT, DIGITAL_INPUT, DIGITAL_INPUT_DIAG, DIGITAL_OUTPUT, DIGITAL_OUTPUT_DIAG, DIGITAL_INOUT, DIGITAL_INOUT_DIAG, DIGITAL_DIAG:
		TerminalManager.RegisterModuleAtTerminal(GVL_SmartCoupler.aDUT_ModuleInterface[usiModuleIndex].FbModuleProcessInputsOutputs,I_Terminal);
		GVL_SmartCoupler.aDUT_ModuleDataAccess[usiModuleIndex].uiModulePiInputSize := GVL_SmartCoupler.aDUT_ModuleInterface[usiModuleIndex].FbModuleProcessInputsOutputs.GetModuleInputSize();
		GVL_SmartCoupler.aDUT_ModuleDataAccess[usiModuleIndex].uiModulePiOutputSize := GVL_SmartCoupler.aDUT_ModuleInterface[usiModuleIndex].FbModuleProcessInputsOutputs.GetModuleOutputSize();

END_CASE
END_ACTION

ACTION DriveDaliModuleAccess:

GVL_SmartCoupler.aDUT_ModuleFunctionAccess[usiModuleIndex].FbDaliMaster(
	bPortDALI	:= GVL_SmartCoupler.bModule647Index, 
	I_Port		:= GVL_SmartCoupler.aDUT_ModuleInterface[usiModuleIndex].FbModule_753_647);

PrgDaliConfigurator();

GVL_SmartCoupler.aDUT_ModuleFunctionAccess[usiModuleIndex].FbDaliSendDimValue.typBallast.bAddress := WORD_TO_BYTE(GVL_SmartCoupler.aDUT_ModuleDataAccess[usiModuleIndex].pawModuleOutput^[1]);
GVL_SmartCoupler.aDUT_ModuleFunctionAccess[usiModuleIndex].FbDaliSendDimValue.typBallast.bPortDALI := GVL_SmartCoupler.bModule647Index;
GVL_SmartCoupler.aDUT_ModuleFunctionAccess[usiModuleIndex].FbDaliSendDimValue.rDimValue := WORD_TO_REAL(GVL_SmartCoupler.aDUT_ModuleDataAccess[usiModuleIndex].pawModuleOutput^[2]);
GVL_SmartCoupler.aDUT_ModuleFunctionAccess[usiModuleIndex].FbDaliSendDimValue();
GVL_SmartCoupler.aDUT_ModuleDataAccess[usiModuleIndex].pawModuleInput^[1] := REAL_TO_WORD(GVL_SmartCoupler.aDUT_ModuleFunctionAccess[usiModuleIndex].FbDaliSendDimValue.rActualLevel);
END_ACTION

ACTION DriveSimpleAIOModuleAccess:

IF (GVL_SmartCoupler.aDUT_ModuleDataAccess[usiModuleIndex].uiModulePiOutputSize > 0) THEN
	GVL_SmartCoupler.aDUT_ModuleInterface[usiModuleIndex].FbModuleProcessInputsOutputs.SetProcessOutData(
		pOutData	:= GVL_SmartCoupler.aDUT_ModuleDataAccess[usiModuleIndex].pawModuleOutput,
		uiNOutData	:= GVL_SmartCoupler.aDUT_ModuleDataAccess[usiModuleIndex].uiModulePiOutputSize);
END_IF

IF (GVL_SmartCoupler.aDUT_ModuleDataAccess[usiModuleIndex].uiModulePiInputSize > 0) THEN
	GVL_SmartCoupler.aDUT_ModuleInterface[usiModuleIndex].FbModuleProcessInputsOutputs.GetProcessInData(
		pInData		:= GVL_SmartCoupler.aDUT_ModuleDataAccess[usiModuleIndex].pawModuleInput,
		uiNInData	:= GVL_SmartCoupler.aDUT_ModuleDataAccess[usiModuleIndex].uiModulePiInputSize);
END_IF
END_ACTION

ACTION DriveKnxModuleAccess:

GVL_SmartCoupler.aDUT_ModuleFunctionAccess[usiModuleIndex].FbKnxMaster_TM.stPhyAddress (*:= GVL_SmartCoupler.aDUT_ModuleDataAccess[usiModuleIndex].pawModuleOutput^[1]*);
GVL_SmartCoupler.aDUT_ModuleFunctionAccess[usiModuleIndex].FbKnxMaster_TM.xFilter_Mode (*:= GVL_SmartCoupler.aDUT_ModuleDataAccess[usiModuleIndex].pawModuleOutput^[2]*);

GVL_SmartCoupler.aDUT_ModuleFunctionAccess[usiModuleIndex].FbKnxMaster_TM(
	bPortKNX	:= GVL_SmartCoupler.bModule646Index, 
	I_Port		:= GVL_SmartCoupler.aDUT_ModuleInterface[usiModuleIndex].FbModule_753_646);

GVL_SmartCoupler.aDUT_ModuleDataAccess[usiModuleIndex].pawModuleInput^[1];
END_ACTION

END_PROGRAM

// PFCx00_SmartCoupler/PFCx00_SmartCoupler/Visualization
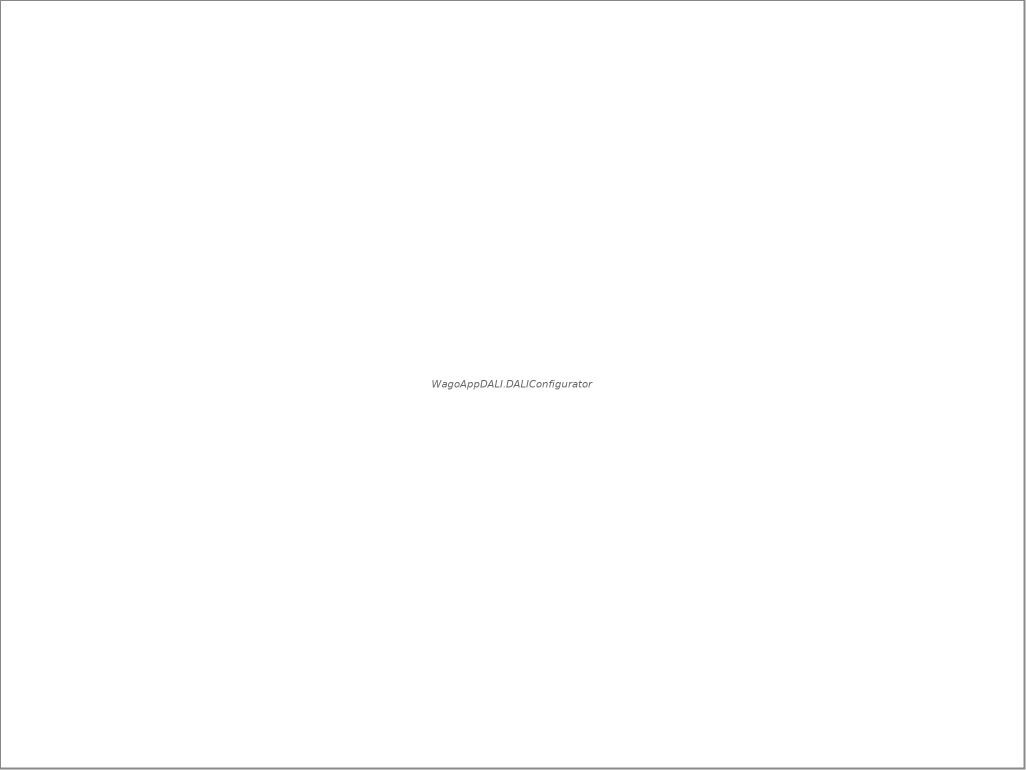
VISUALIZATION Visualization  // 1026x770
    Frame (0,0 1024x768)
        shows WagoAppDALI.DALIConfigurator()
END_VISUALIZATION
